LIN {X 0,Y 118.169,Z 614.006,A -85,B 0,C 180,E1 -30059.995,E2 -30059.995} C_VEL
LIN {X 0,Y 117.877,Z 614.865,A -85,B 0,C 180,E1 -30059.712,E2 -30059.712} C_VEL
LIN {X 0,Y 113.586,Z 625.245,A -85,B 0,C 180,E1 -30059.502,E2 -30059.502} C_VEL
LIN {X 0,Y 107.189,Z 637.349,A -85,B 0,C 180,E1 -30059.098,E2 -30059.098} C_VEL
LIN {X 0,Y 99.298,Z 648.743,A -85,B 0,C 180,E1 -30058.635,E2 -30058.635} C_VEL
LIN {X 0,Y 93.168,Z 656.159,A -85,B 0,C 180,E1 -30058.165,E2 -30058.165} C_VEL
LIN {X 0,Y 84.422,Z 664.947,A -85,B 0,C 180,E1 -30057.397,E2 -30057.397} C_VEL
LIN {X 0,Y 77.444,Z 670.933,A -85,B 0,C 180,E1 -30056.595,E2 -30056.595} C_VEL
LIN {X 0,Y 68.747,Z 677.24,A -85,B 0,C 180,E1 -30055.367,E2 -30055.367} C_VEL
LIN {X 0,Y 59.764,Z 682.696,A -85,B 0,C 180,E1 -30053.548,E2 -30053.548} C_VEL
LIN {X 0,Y 49.831,Z 687.613,A -85,B 0,C 180,E1 -30050.836,E2 -30050.836} C_VEL
LIN {X 0,Y 39.702,Z 691.58,A -85,B 0,C 180,E1 -30046.802,E2 -30046.802} C_VEL
LIN {X 0,Y 29.884,Z 694.52,A -85,B 0,C 180,E1 -30040.167,E2 -30040.167} C_VEL
LIN {X 0,Y 23.763,Z 696.03,A -85,B 0,C 180,E1 -30032.531,E2 -30032.531} C_VEL
LIN {X 0,Y 14.258,Z 697.578,A -85,B 0,C 180,E1 -29999.533,E2 -29999.533} C_VEL
LIN {X 0,Y 12.869,Z 697.867,A -85,B 0,C 180,E1 -29970,E2 -29970} C_VEL
LIN {X 0,Y 18.308,Z 696.97,A -85,B 0,C 180,E1 -29919.849,E2 -29919.849} C_VEL
LIN {X 0,Y 23.763,Z 696.03,A -85,B 0,C 180,E1 -29907.469,E2 -29907.469} C_VEL
LIN {X 0,Y 36.383,Z 692.67,A -85,B 0,C 180,E1 -29895.024,E2 -29895.024} C_VEL
LIN {X 0,Y 46.427,Z 689.041,A -85,B 0,C 180,E1 -29890.284,E2 -29890.284} C_VEL
LIN {X 0,Y 54.933,Z 685.21,A -85,B 0,C 180,E1 -29887.605,E2 -29887.605} C_VEL
LIN {X 0,Y 63.552,Z 680.518,A -85,B 0,C 180,E1 -29885.579,E2 -29885.579} C_VEL
LIN {X 0,Y 72.219,Z 674.865,A -85,B 0,C 180,E1 -29884.083,E2 -29884.083} C_VEL
LIN {X 0,Y 80.93,Z 668.066,A -85,B 0,C 180,E1 -29882.979,E2 -29882.979} C_VEL
LIN {X 0,Y 89.665,Z 659.854,A -85,B 0,C 180,E1 -29882.079,E2 -29882.079} C_VEL
LIN {X 0,Y 96.669,Z 652.036,A -85,B 0,C 180,E1 -29881.551,E2 -29881.551} C_VEL
LIN {X 0,Y 102.804,Z 643.959,A -85,B 0,C 180,E1 -29881.136,E2 -29881.136} C_VEL
LIN {X 0,Y 108.944,Z 634.208,A -85,B 0,C 180,E1 -29880.826,E2 -29880.826} C_VEL
LIN {X 0,Y 114.037,Z 624.239,A -85,B 0,C 180,E1 -29880.518,E2 -29880.518} C_VEL
LIN {X 0,Y 117.877,Z 614.869,A -85,B 0,C 180,E1 -29880.322,E2 -29880.322} C_VEL
LIN {X 0,Y 118.172,Z 613.998,A -85,B 0,C 180,E1 -29880.005,E2 -29880.005} C_VEL
LIN {X 0,Y 117.763,Z 615.989,A -85,B 0,C 180,E1 -29875.422,E2 -29875.422} C_VEL
LIN {X 0,Y 117.614,Z 617.596,A -85,B 0,C 180,E1 -29873.142,E2 -29873.142} C_VEL
LIN {X 0,Y 117.105,Z 620.39,A -85,B 0,C 180,E1 -29870.506,E2 -29870.506} C_VEL
LIN {X 0,Y 116.14,Z 624.865,A -85,B 0,C 180,E1 -29867.601,E2 -29867.601} C_VEL
LIN {X 0,Y 115.107,Z 628.526,A -85,B 0,C 180,E1 -29865.87,E2 -29865.87} C_VEL
LIN {X 0,Y 111.487,Z 638.971,A -85,B 0,C 180,E1 -29861.01,E2 -29861.01} C_VEL
LIN {X 0,Y 108.455,Z 647.592,A -85,B 0,C 180,E1 -29856.115,E2 -29856.115} C_VEL
LIN {X 0,Y 106.01,Z 655.467,A -85,B 0,C 180,E1 -29850.569,E2 -29850.569} C_VEL
LIN {X 0,Y 104.558,Z 661.545,A -85,B 0,C 180,E1 -29845.542,E2 -29845.542} C_VEL
LIN {X 0,Y 103.809,Z 669.53,A -85,B 0,C 180,E1 -29837.398,E2 -29837.398} C_VEL
LIN {X 0,Y 104.443,Z 673.875,A -85,B 0,C 180,E1 -29832.262,E2 -29832.262} C_VEL
LIN {X 0,Y 106.959,Z 679.238,A -85,B 0,C 180,E1 -29824.795,E2 -29824.795} C_VEL
LIN {X 0,Y 112.881,Z 684.586,A -85,B 0,C 180,E1 -29815.837,E2 -29815.837} C_VEL
LIN {X 0,Y 119.382,Z 687.768,A -85,B 0,C 180,E1 -29809.642,E2 -29809.642} C_VEL
LIN {X 0,Y 130.255,Z 690.725,A -85,B 0,C 180,E1 -29802.464,E2 -29802.464} C_VEL
LIN {X 0,Y 141.656,Z 692.301,A -85,B 0,C 180,E1 -29797.174,E2 -29797.174} C_VEL
LIN {X 0,Y 154.94,Z 692.973,A -85,B 0,C 180,E1 -29792.6,E2 -29792.6} C_VEL
LIN {X 0,Y 164.279,Z 692.971,A -85,B 0,C 180,E1 -29790,E2 -29790} C_VEL
LIN {X 0,Y 146.004,Z 692.638,A -85,B 0,C 180,E1 -29784.476,E2 -29784.476} C_VEL
LIN {X 0,Y 135.499,Z 691.643,A -85,B 0,C 180,E1 -29780.195,E2 -29780.195} C_VEL
LIN {X 0,Y 129.979,Z 690.679,A -85,B 0,C 180,E1 -29777.394,E2 -29777.394} C_VEL
LIN {X 0,Y 125.959,Z 690.113,A -85,B 0,C 180,E1 -29775.472,E2 -29775.472} C_VEL
LIN {X 0,Y 112.356,Z 688.655,A -85,B 0,C 180,E1 -29769.954,E2 -29769.954} C_VEL
LIN {X 0,Y 108.7,Z 687.726,A -85,B 0,C 180,E1 -29767.606,E2 -29767.606} C_VEL
LIN {X 0,Y 107.751,Z 687.318,A -85,B 0,C 180,E1 -29766.722,E2 -29766.722} C_VEL
LIN {X 0,Y 102.213,Z 683.666,A -85,B 0,C 180,E1 -29759.228,E2 -29759.228} C_VEL
LIN {X 0,Y 98.445,Z 678.262,A -85,B 0,C 180,E1 -29750.021,E2 -29750.021} C_VEL
LIN {X 0,Y 97.481,Z 673.186,A -85,B 0,C 180,E1 -29742.695,E2 -29742.695} C_VEL
LIN {X 0,Y 98.282,Z 666.575,A -85,B 0,C 180,E1 -29734.887,E2 -29734.887} C_VEL
LIN {X 0,Y 100.458,Z 659.553,A -85,B 0,C 180,E1 -29728.17,E2 -29728.17} C_VEL
LIN {X 0,Y 103.759,Z 651.316,A -85,B 0,C 180,E1 -29721.863,E2 -29721.863} C_VEL
LIN {X 0,Y 107.51,Z 642.683,A -85,B 0,C 180,E1 -29716.593,E2 -29716.593} C_VEL
LIN {X 0,Y 111.381,Z 633.584,A -85,B 0,C 180,E1 -29712.125,E2 -29712.125} C_VEL
LIN {X 0,Y 112.591,Z 630.569,A -85,B 0,C 180,E1 -29710.787,E2 -29710.787} C_VEL
LIN {X 0,Y 113.778,Z 627.253,A -85,B 0,C 180,E1 -29708.772,E2 -29708.772} C_VEL
LIN {X 0,Y 114.375,Z 624.991,A -85,B 0,C 180,E1 -29707.054,E2 -29707.054} C_VEL
LIN {X 0,Y 114.764,Z 623.365,A -85,B 0,C 180,E1 -29705.265,E2 -29705.265} C_VEL
LIN {X 0,Y 115.055,Z 622.207,A -85,B 0,C 180,E1 -29703.497,E2 -29703.497} C_VEL
LIN {X 0,Y 114.198,Z 624.038,A -85,B 0,C 180,E1 -29703.082,E2 -29703.082} C_VEL
LIN {X 0,Y 109.96,Z 632.42,A -85,B 0,C 180,E1 -29702.978,E2 -29702.978} C_VEL
LIN {X 0,Y 104.67,Z 641.139,A -85,B 0,C 180,E1 -29702.856,E2 -29702.856} C_VEL
LIN {X 0,Y 98.501,Z 649.644,A -85,B 0,C 180,E1 -29702.715,E2 -29702.715} C_VEL
LIN {X 0,Y 91.451,Z 657.81,A -85,B 0,C 180,E1 -29702.514,E2 -29702.514} C_VEL
LIN {X 0,Y 84.399,Z 664.75,A -85,B 0,C 180,E1 -29702.236,E2 -29702.236} C_VEL
LIN {X 0,Y 77.349,Z 670.736,A -85,B 0,C 180,E1 -29701.877,E2 -29701.877} C_VEL
LIN {X 0,Y 68.54,Z 677.044,A -85,B 0,C 180,E1 -29701.309,E2 -29701.309} C_VEL
LIN {X 0,Y 59.739,Z 682.319,A -85,B 0,C 180,E1 -29700.453,E2 -29700.453} C_VEL
LIN {X 0,Y 49.202,Z 687.416,A -85,B 0,C 180,E1 -29699.067,E2 -29699.067} C_VEL
LIN {X 0,Y 38.701,Z 691.383,A -85,B 0,C 180,E1 -29697.149,E2 -29697.149} C_VEL
LIN {X 0,Y 28.273,Z 694.323,A -85,B 0,C 180,E1 -29693.877,E2 -29693.877} C_VEL
LIN {X 0,Y 21.426,Z 695.833,A -85,B 0,C 180,E1 -29689.747,E2 -29689.747} C_VEL
LIN {X 0,Y 8.799,Z 697.381,A -85,B 0,C 180,E1 -29663.004,E2 -29663.004} C_VEL
LIN {X 0,Y 5.756,Z 697.671,A -85,B 0,C 180,E1 -29610,E2 -29610} C_VEL
LIN {X 0,Y 14.791,Z 696.773,A -85,B 0,C 180,E1 -29538.136,E2 -29538.136} C_VEL
LIN {X 0,Y 21.426,Z 695.833,A -85,B 0,C 180,E1 -29530.252,E2 -29530.252} C_VEL
LIN {X 0,Y 35.216,Z 692.474,A -85,B 0,C 180,E1 -29523.768,E2 -29523.768} C_VEL
LIN {X 0,Y 45.697,Z 688.844,A -85,B 0,C 180,E1 -29521.471,E2 -29521.471} C_VEL
LIN {X 0,Y 56.223,Z 684.109,A -85,B 0,C 180,E1 -29519.932,E2 -29519.932} C_VEL
LIN {X 0,Y 66.779,Z 678.135,A -85,B 0,C 180,E1 -29518.818,E2 -29518.818} C_VEL
LIN {X 0,Y 75.587,Z 672.046,A -85,B 0,C 180,E1 -29518.198,E2 -29518.198} C_VEL
LIN {X 0,Y 82.636,Z 666.31,A -85,B 0,C 180,E1 -29517.859,E2 -29517.859} C_VEL
LIN {X 0,Y 89.689,Z 659.658,A -85,B 0,C 180,E1 -29517.539,E2 -29517.539} C_VEL
LIN {X 0,Y 96.738,Z 651.84,A -85,B 0,C 180,E1 -29517.345,E2 -29517.345} C_VEL
LIN {X 0,Y 102.908,Z 643.763,A -85,B 0,C 180,E1 -29517.185,E2 -29517.185} C_VEL
LIN {X 0,Y 109.074,Z 634.012,A -85,B 0,C 180,E1 -29517.087,E2 -29517.087} C_VEL
LIN {X 0,Y 114.221,Z 623.981,A -85,B 0,C 180,E1 -29516.957,E2 -29516.957} C_VEL
LIN {X 0,Y 114.699,Z 622.913,A -85,B 0,C 180,E1 -29516.954,E2 -29516.954} C_VEL
LIN {X 0,Y 115.069,Z 622.175,A -85,B 0,C 180,E1 -29516.504,E2 -29516.504} C_VEL
LIN {X 0,Y 114.776,Z 623.339,A -85,B 0,C 180,E1 -29514.735,E2 -29514.735} C_VEL
LIN {X 0,Y 114.111,Z 626.031,A -85,B 0,C 180,E1 -29512.084,E2 -29512.084} C_VEL
LIN {X 0,Y 113.261,Z 628.786,A -85,B 0,C 180,E1 -29510.225,E2 -29510.225} C_VEL
LIN {X 0,Y 111.785,Z 632.565,A -85,B 0,C 180,E1 -29508.324,E2 -29508.324} C_VEL
LIN {X 0,Y 108.15,Z 641.164,A -85,B 0,C 180,E1 -29504.221,E2 -29504.221} C_VEL
LIN {X 0,Y 104.826,Z 648.774,A -85,B 0,C 180,E1 -29499.82,E2 -29499.82} C_VEL
LIN {X 0,Y 102.329,Z 654.783,A -85,B 0,C 180,E1 -29495.671,E2 -29495.671} C_VEL
LIN {X 0,Y 99.693,Z 661.815,A -85,B 0,C 180,E1 -29489.833,E2 -29489.833} C_VEL
LIN {X 0,Y 97.787,Z 669.151,A -85,B 0,C 180,E1 -29482.238,E2 -29482.238} C_VEL
LIN {X 0,Y 97.688,Z 675.553,A -85,B 0,C 180,E1 -29474.002,E2 -29474.002} C_VEL
LIN {X 0,Y 99.545,Z 680.564,A -85,B 0,C 180,E1 -29466.239,E2 -29466.239} C_VEL
LIN {X 0,Y 103.704,Z 684.913,A -85,B 0,C 180,E1 -29458.25,E2 -29458.25} C_VEL
LIN {X 0,Y 108.04,Z 687.465,A -85,B 0,C 180,E1 -29452.973,E2 -29452.973} C_VEL
LIN {X 0,Y 116.689,Z 690.455,A -85,B 0,C 180,E1 -29445.517,E2 -29445.517} C_VEL
LIN {X 0,Y 128.026,Z 692.417,A -85,B 0,C 180,E1 -29438.879,E2 -29438.879} C_VEL
LIN {X 0,Y 143.096,Z 693.294,A -85,B 0,C 180,E1 -29432.815,E2 -29432.815} C_VEL
LIN {X 0,Y 152.364,Z 693.301,A -85,B 0,C 180,E1 -29430,E2 -29430} C_VEL
LIN {X 0,Y 140.823,Z 693.282,A -85,B 0,C 180,E1 -29426.413,E2 -29426.413} C_VEL
LIN {X 0,Y 126.564,Z 692.278,A -85,B 0,C 180,E1 -29420.411,E2 -29420.411} C_VEL
LIN {X 0,Y 116.678,Z 690.465,A -85,B 0,C 180,E1 -29414.503,E2 -29414.503} C_VEL
LIN {X 0,Y 107.751,Z 687.318,A -85,B 0,C 180,E1 -29406.722,E2 -29406.722} C_VEL
LIN {X 0,Y 104.734,Z 686.184,A -85,B 0,C 180,E1 -29404.045,E2 -29404.045} C_VEL
LIN {X 0,Y 94.611,Z 683.451,A -85,B 0,C 180,E1 -29395.741,E2 -29395.741} C_VEL
LIN {X 0,Y 92.503,Z 682.035,A -85,B 0,C 180,E1 -29392.488,E2 -29392.488} C_VEL
LIN {X 0,Y 92.124,Z 681.457,A -85,B 0,C 180,E1 -29391.348,E2 -29391.348} C_VEL
LIN {X 0,Y 91.057,Z 677.2,A -85,B 0,C 180,E1 -29383.988,E2 -29383.988} C_VEL
LIN {X 0,Y 91.647,Z 671.97,A -85,B 0,C 180,E1 -29376.453,E2 -29376.453} C_VEL
LIN {X 0,Y 93.783,Z 665.721,A -85,B 0,C 180,E1 -29369.14,E2 -29369.14} C_VEL
LIN {X 0,Y 96.531,Z 659.898,A -85,B 0,C 180,E1 -29363.595,E2 -29363.595} C_VEL
LIN {X 0,Y 100.499,Z 652.251,A -85,B 0,C 180,E1 -29357.733,E2 -29357.733} C_VEL
LIN {X 0,Y 104.974,Z 643.783,A -85,B 0,C 180,E1 -29352.617,E2 -29352.617} C_VEL
LIN {X 0,Y 109.775,Z 634.122,A -85,B 0,C 180,E1 -29347.933,E2 -29347.933} C_VEL
LIN {X 0,Y 110.243,Z 633.033,A -85,B 0,C 180,E1 -29347.319,E2 -29347.319} C_VEL
LIN {X 0,Y 109.183,Z 634.691,A -85,B 0,C 180,E1 -29346.655,E2 -29346.655} C_VEL
LIN {X 0,Y 101.738,Z 646.132,A -85,B 0,C 180,E1 -29346.782,E2 -29346.782} C_VEL
LIN {X 0,Y 93.799,Z 655.765,A -85,B 0,C 180,E1 -29346.899,E2 -29346.899} C_VEL
LIN {X 0,Y 84.976,Z 664.553,A -85,B 0,C 180,E1 -29347.041,E2 -29347.041} C_VEL
LIN {X 0,Y 77.909,Z 670.539,A -85,B 0,C 180,E1 -29347.126,E2 -29347.126} C_VEL
LIN {X 0,Y 69.072,Z 676.846,A -85,B 0,C 180,E1 -29347.236,E2 -29347.236} C_VEL
LIN {X 0,Y 60.223,Z 682.121,A -85,B 0,C 180,E1 -29347.28,E2 -29347.28} C_VEL
LIN {X 0,Y 49.602,Z 687.219,A -85,B 0,C 180,E1 -29347.337,E2 -29347.337} C_VEL
LIN {X 0,Y 39.005,Z 691.185,A -85,B 0,C 180,E1 -29347.697,E2 -29347.697} C_VEL
LIN {X 0,Y 28.409,Z 694.126,A -85,B 0,C 180,E1 -29348.301,E2 -29348.301} C_VEL
LIN {X 0,Y 21.345,Z 695.635,A -85,B 0,C 180,E1 -29348.978,E2 -29348.978} C_VEL
LIN {X 0,Y 7.264,Z 697.184,A -85,B 0,C 180,E1 -29354.645,E2 -29354.645} C_VEL
LIN {X 0,Y 1.343,Z 697.475,A -85,B 0,C 180,E1 -29430,E2 -29430} C_VEL
LIN {X 0,Y 14.283,Z 696.575,A -85,B 0,C 180,E1 -29509.759,E2 -29509.759} C_VEL
LIN {X 0,Y 21.345,Z 695.635,A -85,B 0,C 180,E1 -29511.022,E2 -29511.022} C_VEL
LIN {X 0,Y 35.466,Z 692.277,A -85,B 0,C 180,E1 -29512.216,E2 -29512.216} C_VEL
LIN {X 0,Y 46.066,Z 688.647,A -85,B 0,C 180,E1 -29512.589,E2 -29512.589} C_VEL
LIN {X 0,Y 55.231,Z 684.646,A -85,B 0,C 180,E1 -29512.701,E2 -29512.701} C_VEL
LIN {X 0,Y 65.538,Z 679.03,A -85,B 0,C 180,E1 -29512.713,E2 -29512.713} C_VEL
LIN {X 0,Y 74.378,Z 673.16,A -85,B 0,C 180,E1 -29512.813,E2 -29512.813} C_VEL
LIN {X 0,Y 81.441,Z 667.673,A -85,B 0,C 180,E1 -29512.927,E2 -29512.927} C_VEL
LIN {X 0,Y 90.272,Z 659.462,A -85,B 0,C 180,E1 -29513.035,E2 -29513.035} C_VEL
LIN {X 0,Y 97.326,Z 651.643,A -85,B 0,C 180,E1 -29513.161,E2 -29513.161} C_VEL
LIN {X 0,Y 103.498,Z 643.567,A -85,B 0,C 180,E1 -29513.262,E2 -29513.262} C_VEL
LIN {X 0,Y 109.172,Z 634.704,A -85,B 0,C 180,E1 -29513.368,E2 -29513.368} C_VEL
LIN {X 0,Y 110.22,Z 633.075,A -85,B 0,C 180,E1 -29512.679,E2 -29512.679} C_VEL
LIN {X 0,Y 107.201,Z 639.436,A -85,B 0,C 180,E1 -29509.539,E2 -29509.539} C_VEL
LIN {X 0,Y 102.878,Z 647.758,A -85,B 0,C 180,E1 -29505.104,E2 -29505.104} C_VEL
LIN {X 0,Y 99.152,Z 654.795,A -85,B 0,C 180,E1 -29500.508,E2 -29500.508} C_VEL
LIN {X 0,Y 95.086,Z 662.884,A -85,B 0,C 180,E1 -29493.682,E2 -29493.682} C_VEL
LIN {X 0,Y 92.412,Z 669.407,A -85,B 0,C 180,E1 -29486.777,E2 -29486.777} C_VEL
LIN {X 0,Y 91.145,Z 675.365,A -85,B 0,C 180,E1 -29478.846,E2 -29478.846} C_VEL
LIN {X 0,Y 91.811,Z 680.718,A -85,B 0,C 180,E1 -29470.061,E2 -29470.061} C_VEL
LIN {X 0,Y 94.843,Z 685.153,A -85,B 0,C 180,E1 -29461.245,E2 -29461.245} C_VEL
LIN {X 0,Y 99.773,Z 688.355,A -85,B 0,C 180,E1 -29453.709,E2 -29453.709} C_VEL
LIN {X 0,Y 109.071,Z 691.344,A -85,B 0,C 180,E1 -29444.891,E2 -29444.891} C_VEL
LIN {X 0,Y 115.719,Z 692.583,A -85,B 0,C 180,E1 -29440.498,E2 -29440.498} C_VEL
LIN {X 0,Y 126.949,Z 693.553,A -85,B 0,C 180,E1 -29434.865,E2 -29434.865} C_VEL
LIN {X 0,Y 140.481,Z 693.629,A -85,B 0,C 180,E1 -29430,E2 -29430} C_VEL
LIN {X 0,Y 126.947,Z 693.555,A -85,B 0,C 180,E1 -29425.143,E2 -29425.143} C_VEL
LIN {X 0,Y 114.594,Z 692.424,A -85,B 0,C 180,E1 -29418.861,E2 -29418.861} C_VEL
LIN {X 0,Y 103.287,Z 689.725,A -85,B 0,C 180,E1 -29410.11,E2 -29410.11} C_VEL
LIN {X 0,Y 98.564,Z 687.752,A -85,B 0,C 180,E1 -29404.671,E2 -29404.671} C_VEL
LIN {X 0,Y 93.554,Z 683.757,A -85,B 0,C 180,E1 -29395.713,E2 -29395.713} C_VEL
LIN {X 0,Y 92.124,Z 681.457,A -85,B 0,C 180,E1 -29391.348,E2 -29391.348} C_VEL
LIN {X 0,Y 90.843,Z 679.857,A -85,B 0,C 180,E1 -29387.872,E2 -29387.872} C_VEL
LIN {X 0,Y 86.151,Z 675.628,A -85,B 0,C 180,E1 -29377.053,E2 -29377.053} C_VEL
LIN {X 0,Y 86,Z 673.585,A -85,B 0,C 180,E1 -29373.388,E2 -29373.388} C_VEL
LIN {X 0,Y 86.266,Z 672.75,A -85,B 0,C 180,E1 -29372.221,E2 -29372.221} C_VEL
LIN {X 0,Y 89.365,Z 666.65,A -85,B 0,C 180,E1 -29364.808,E2 -29364.808} C_VEL
LIN {X 0,Y 93.127,Z 660.513,A -85,B 0,C 180,E1 -29358.914,E2 -29358.914} C_VEL
LIN {X 0,Y 98.879,Z 651.385,A -85,B 0,C 180,E1 -29352.234,E2 -29352.234} C_VEL
LIN {X 0,Y 100.187,Z 649.251,A -85,B 0,C 180,E1 -29350.867,E2 -29350.867} C_VEL
LIN {X 0,Y 93.162,Z 657.417,A -85,B 0,C 180,E1 -29351.278,E2 -29351.278} C_VEL
LIN {X 0,Y 86.139,Z 664.356,A -85,B 0,C 180,E1 -29351.747,E2 -29351.747} C_VEL
LIN {X 0,Y 79.108,Z 670.342,A -85,B 0,C 180,E1 -29352.248,E2 -29352.248} C_VEL
LIN {X 0,Y 70.325,Z 676.65,A -85,B 0,C 180,E1 -29353.002,E2 -29353.002} C_VEL
LIN {X 0,Y 61.537,Z 681.924,A -85,B 0,C 180,E1 -29353.892,E2 -29353.892} C_VEL
LIN {X 0,Y 51.01,Z 687.021,A -85,B 0,C 180,E1 -29355.327,E2 -29355.327} C_VEL
LIN {X 0,Y 40.584,Z 690.988,A -85,B 0,C 180,E1 -29357.742,E2 -29357.742} C_VEL
LIN {X 0,Y 30.266,Z 693.93,A -85,B 0,C 180,E1 -29361.747,E2 -29361.747} C_VEL
LIN {X 0,Y 23.541,Z 695.438,A -85,B 0,C 180,E1 -29366.414,E2 -29366.414} C_VEL
LIN {X 0,Y 11.387,Z 696.987,A -85,B 0,C 180,E1 -29391.89,E2 -29391.89} C_VEL
LIN {X 0,Y 8.433,Z 697.279,A -85,B 0,C 180,E1 -29430,E2 -29430} C_VEL
LIN {X 0,Y 17.064,Z 696.378,A -85,B 0,C 180,E1 -29485.457,E2 -29485.457} C_VEL
LIN {X 0,Y 23.542,Z 695.438,A -85,B 0,C 180,E1 -29493.585,E2 -29493.585} C_VEL
LIN {X 0,Y 37.113,Z 692.08,A -85,B 0,C 180,E1 -29501.231,E2 -29501.231} C_VEL
LIN {X 0,Y 47.512,Z 688.451,A -85,B 0,C 180,E1 -29504.046,E2 -29504.046} C_VEL
LIN {X 0,Y 55.54,Z 684.983,A -85,B 0,C 180,E1 -29505.352,E2 -29505.352} C_VEL
LIN {X 0,Y 66.815,Z 678.834,A -85,B 0,C 180,E1 -29506.646,E2 -29506.646} C_VEL
LIN {X 0,Y 75.601,Z 672.963,A -85,B 0,C 180,E1 -29507.444,E2 -29507.444} C_VEL
LIN {X 0,Y 82.617,Z 667.476,A -85,B 0,C 180,E1 -29508.032,E2 -29508.032} C_VEL
LIN {X 0,Y 91.409,Z 659.265,A -85,B 0,C 180,E1 -29508.6,E2 -29508.6} C_VEL
LIN {X 0,Y 98.427,Z 651.447,A -85,B 0,C 180,E1 -29509.046,E2 -29509.046} C_VEL
LIN {X 0,Y 100.215,Z 649.247,A -85,B 0,C 180,E1 -29509.05,E2 -29509.05} C_VEL
LIN {X 0,Y 95.856,Z 656.134,A -85,B 0,C 180,E1 -29504.553,E2 -29504.553} C_VEL
LIN {X 0,Y 90.993,Z 663.897,A -85,B 0,C 180,E1 -29497.947,E2 -29497.947} C_VEL
LIN {X 0,Y 87.501,Z 670.11,A -85,B 0,C 180,E1 -29491.198,E2 -29491.198} C_VEL
LIN {X 0,Y 85.508,Z 674.843,A -85,B 0,C 180,E1 -29484.886,E2 -29484.886} C_VEL
LIN {X 0,Y 84.56,Z 680.62,A -85,B 0,C 180,E1 -29475.064,E2 -29475.064} C_VEL
LIN {X 0,Y 86.454,Z 685.429,A -85,B 0,C 180,E1 -29464.683,E2 -29464.683} C_VEL
LIN {X 0,Y 89.357,Z 688.037,A -85,B 0,C 180,E1 -29458.158,E2 -29458.158} C_VEL
LIN {X 0,Y 96.479,Z 691.081,A -85,B 0,C 180,E1 -29448.762,E2 -29448.762} C_VEL
LIN {X 0,Y 107.096,Z 693.104,A -85,B 0,C 180,E1 -29440.186,E2 -29440.186} C_VEL
LIN {X 0,Y 120.064,Z 693.922,A -85,B 0,C 180,E1 -29433.356,E2 -29433.356} C_VEL
LIN {X 0,Y 128.809,Z 693.952,A -85,B 0,C 180,E1 -29430,E2 -29430} C_VEL
LIN {X 0,Y 113.19,Z 693.668,A -85,B 0,C 180,E1 -29423.383,E2 -29423.383} C_VEL
LIN {X 0,Y 104.921,Z 692.887,A -85,B 0,C 180,E1 -29418.408,E2 -29418.408} C_VEL
LIN {X 0,Y 96.479,Z 691.081,A -85,B 0,C 180,E1 -29411.237,E2 -29411.237} C_VEL
LIN {X 0,Y 88.743,Z 687.517,A -85,B 0,C 180,E1 -29400.577,E2 -29400.577} C_VEL
LIN {X 0,Y 85.418,Z 683.748,A -85,B 0,C 180,E1 -29391.394,E2 -29391.394} C_VEL
LIN {X 0,Y 84.572,Z 678.795,A -85,B 0,C 180,E1 -29381.592,E2 -29381.592} C_VEL
LIN {X 0,Y 86.266,Z 672.75,A -85,B 0,C 180,E1 -29372.221,E2 -29372.221} C_VEL
LIN {X 0,Y 86.512,Z 671.274,A -85,B 0,C 180,E1 -29369.764,E2 -29369.764} C_VEL
LIN {X 0,Y 85.588,Z 667.944,A -85,B 0,C 180,E1 -29361.065,E2 -29361.065} C_VEL
LIN {X 0,Y 86.473,Z 666.237,A -85,B 0,C 180,E1 -29358.738,E2 -29358.738} C_VEL
LIN {X 0,Y 88.039,Z 664.142,A -85,B 0,C 180,E1 -29356.68,E2 -29356.68} C_VEL
LIN {X 0,Y 87.862,Z 664.16,A -85,B 0,C 180,E1 -29356.289,E2 -29356.289} C_VEL
LIN {X 0,Y 80.916,Z 670.146,A -85,B 0,C 180,E1 -29357.176,E2 -29357.176} C_VEL
LIN {X 0,Y 72.266,Z 676.452,A -85,B 0,C 180,E1 -29358.524,E2 -29358.524} C_VEL
LIN {X 0,Y 63.633,Z 681.726,A -85,B 0,C 180,E1 -29360.153,E2 -29360.153} C_VEL
LIN {X 0,Y 53.345,Z 686.824,A -85,B 0,C 180,E1 -29362.748,E2 -29362.748} C_VEL
LIN {X 0,Y 43.294,Z 690.79,A -85,B 0,C 180,E1 -29366.77,E2 -29366.77} C_VEL
LIN {X 0,Y 33.556,Z 693.733,A -85,B 0,C 180,E1 -29373.097,E2 -29373.097} C_VEL
LIN {X 0,Y 27.471,Z 695.24,A -85,B 0,C 180,E1 -29379.872,E2 -29379.872} C_VEL
LIN {X 0,Y 17.543,Z 696.791,A -85,B 0,C 180,E1 -29406.384,E2 -29406.384} C_VEL
LIN {X 0,Y 15.542,Z 697.082,A -85,B 0,C 180,E1 -29430,E2 -29430} C_VEL
LIN {X 0,Y 21.908,Z 696.181,A -85,B 0,C 180,E1 -29469.911,E2 -29469.911} C_VEL
LIN {X 0,Y 27.471,Z 695.24,A -85,B 0,C 180,E1 -29480.128,E2 -29480.128} C_VEL
LIN {X 0,Y 39.991,Z 691.882,A -85,B 0,C 180,E1 -29491.484,E2 -29491.484} C_VEL
LIN {X 0,Y 49.95,Z 688.253,A -85,B 0,C 180,E1 -29496.142,E2 -29496.142} C_VEL
LIN {X 0,Y 60.19,Z 683.517,A -85,B 0,C 180,E1 -29499.082,E2 -29499.082} C_VEL
LIN {X 0,Y 70.537,Z 677.545,A -85,B 0,C 180,E1 -29501.178,E2 -29501.178} C_VEL
LIN {X 0,Y 79.19,Z 671.456,A -85,B 0,C 180,E1 -29502.562,E2 -29502.562} C_VEL
LIN {X 0,Y 85.712,Z 666.088,A -85,B 0,C 180,E1 -29503.452,E2 -29503.452} C_VEL
LIN {X 0,Y 87.861,Z 664.16,A -85,B 0,C 180,E1 -29503.712,E2 -29503.712} C_VEL
LIN {X 0,Y 88.039,Z 664.143,A -85,B 0,C 180,E1 -29503.322,E2 -29503.322} C_VEL
LIN {X 0,Y 83.847,Z 669.909,A -85,B 0,C 180,E1 -29497.22,E2 -29497.22} C_VEL
LIN {X 0,Y 79.779,Z 676.411,A -85,B 0,C 180,E1 -29488.102,E2 -29488.102} C_VEL
LIN {X 0,Y 78.039,Z 681.486,A -85,B 0,C 180,E1 -29478.662,E2 -29478.662} C_VEL
LIN {X 0,Y 78.573,Z 685.701,A -85,B 0,C 180,E1 -29468.764,E2 -29468.764} C_VEL
LIN {X 0,Y 81.215,Z 688.752,A -85,B 0,C 180,E1 -29460.093,E2 -29460.093} C_VEL
LIN {X 0,Y 84.533,Z 690.555,A -85,B 0,C 180,E1 -29453.881,E2 -29453.881} C_VEL
LIN {X 0,Y 94.469,Z 693.182,A -85,B 0,C 180,E1 -29442.896,E2 -29442.896} C_VEL
LIN {X 0,Y 108.891,Z 694.232,A -85,B 0,C 180,E1 -29433.7,E2 -29433.7} C_VEL
LIN {X 0,Y 117.313,Z 694.269,A -85,B 0,C 180,E1 -29430,E2 -29430} C_VEL
LIN {X 0,Y 105.853,Z 694.207,A -85,B 0,C 180,E1 -29424.741,E2 -29424.741} C_VEL
LIN {X 0,Y 93.894,Z 693.094,A -85,B 0,C 180,E1 -29416.638,E2 -29416.638} C_VEL
LIN {X 0,Y 84.059,Z 690.299,A -85,B 0,C 180,E1 -29405.289,E2 -29405.289} C_VEL
LIN {X 0,Y 80.697,Z 688.313,A -85,B 0,C 180,E1 -29398.497,E2 -29398.497} C_VEL
LIN {X 0,Y 77.969,Z 683.667,A -85,B 0,C 180,E1 -29386.133,E2 -29386.133} C_VEL
LIN {X 0,Y 78.844,Z 678.402,A -85,B 0,C 180,E1 -29375.283,E2 -29375.283} C_VEL
LIN {X 0,Y 81.805,Z 672.898,A -85,B 0,C 180,E1 -29366.628,E2 -29366.628} C_VEL
LIN {X 0,Y 86.473,Z 666.237,A -85,B 0,C 180,E1 -29358.738,E2 -29358.738} C_VEL
LIN {X 0,Y 85.989,Z 666.47,A -85,B 0,C 180,E1 -29358.239,E2 -29358.239} C_VEL
LIN {X 0,Y 84.009,Z 668.065,A -85,B 0,C 180,E1 -29358.045,E2 -29358.045} C_VEL
LIN {X 0,Y 80.183,Z 671.177,A -85,B 0,C 180,E1 -29358.876,E2 -29358.876} C_VEL
LIN {X 0,Y 74.975,Z 675.481,A -85,B 0,C 180,E1 -29361.196,E2 -29361.196} C_VEL
LIN {X 0,Y 70.97,Z 678.378,A -85,B 0,C 180,E1 -29363.306,E2 -29363.306} C_VEL
LIN {X 0,Y 65.72,Z 681.88,A -85,B 0,C 180,E1 -29365.904,E2 -29365.904} C_VEL
LIN {X 0,Y 62.303,Z 683.739,A -85,B 0,C 180,E1 -29367.227,E2 -29367.227} C_VEL
LIN {X 0,Y 53.234,Z 688.056,A -85,B 0,C 180,E1 -29370.894,E2 -29370.894} C_VEL
LIN {X 0,Y 43.855,Z 691.685,A -85,B 0,C 180,E1 -29376.749,E2 -29376.749} C_VEL
LIN {X 0,Y 32.51,Z 695.043,A -85,B 0,C 180,E1 -29389.569,E2 -29389.569} C_VEL
LIN {X 0,Y 24.25,Z 696.593,A -85,B 0,C 180,E1 -29413.154,E2 -29413.154} C_VEL
LIN {X 0,Y 22.64,Z 696.886,A -85,B 0,C 180,E1 -29430,E2 -29430} C_VEL
LIN {X 0,Y 27.749,Z 695.984,A -85,B 0,C 180,E1 -29460.433,E2 -29460.433} C_VEL
LIN {X 0,Y 32.51,Z 695.043,A -85,B 0,C 180,E1 -29470.431,E2 -29470.431} C_VEL
LIN {X 0,Y 43.855,Z 691.685,A -85,B 0,C 180,E1 -29483.252,E2 -29483.252} C_VEL
LIN {X 0,Y 53.241,Z 688.056,A -85,B 0,C 180,E1 -29489.095,E2 -29489.095} C_VEL
LIN {X 0,Y 61.039,Z 684.426,A -85,B 0,C 180,E1 -29492.32,E2 -29492.32} C_VEL
LIN {X 0,Y 71.598,Z 678.351,A -85,B 0,C 180,E1 -29495.5,E2 -29495.5} C_VEL
LIN {X 0,Y 76.518,Z 675.149,A -85,B 0,C 180,E1 -29496.703,E2 -29496.703} C_VEL
LIN {X 0,Y 72.132,Z 681.778,A -85,B 0,C 180,E1 -29484.236,E2 -29484.236} C_VEL
LIN {X 0,Y 71.225,Z 685.97,A -85,B 0,C 180,E1 -29473.686,E2 -29473.686} C_VEL
LIN {X 0,Y 72.377,Z 688.588,A -85,B 0,C 180,E1 -29465.634,E2 -29465.634} C_VEL
LIN {X 0,Y 76.926,Z 691.599,A -85,B 0,C 180,E1 -29454.013,E2 -29454.013} C_VEL
LIN {X 0,Y 86.343,Z 693.736,A -85,B 0,C 180,E1 -29442.415,E2 -29442.415} C_VEL
LIN {X 0,Y 98.59,Z 694.541,A -85,B 0,C 180,E1 -29433.742,E2 -29433.742} C_VEL
LIN {X 0,Y 106.034,Z 694.581,A -85,B 0,C 180,E1 -29430,E2 -29430} C_VEL
LIN {X 0,Y 90.5,Z 694.175,A -85,B 0,C 180,E1 -29421.065,E2 -29421.065} C_VEL
LIN {X 0,Y 81.208,Z 692.798,A -85,B 0,C 180,E1 -29412.144,E2 -29412.144} C_VEL
LIN {X 0,Y 74.962,Z 690.58,A -85,B 0,C 180,E1 -29402.046,E2 -29402.046} C_VEL
LIN {X 0,Y 71.771,Z 687.685,A -85,B 0,C 180,E1 -29391.556,E2 -29391.556} C_VEL
LIN {X 0,Y 71.375,Z 683.795,A -85,B 0,C 180,E1 -29380.444,E2 -29380.444} C_VEL
LIN {X 0,Y 73.457,Z 679.315,A -85,B 0,C 180,E1 -29370.564,E2 -29370.564} C_VEL
LIN {X 0,Y 76.515,Z 675.149,A -85,B 0,C 180,E1 -29363.292,E2 -29363.292} C_VEL
LIN {X 0,Y 66.422,Z 681.529,A -85,B 0,C 180,E1 -29365.927,E2 -29365.927} C_VEL
LIN {X 0,Y 62.303,Z 683.739,A -85,B 0,C 180,E1 -29367.227,E2 -29367.227} C_VEL
LIN {X 0,Y 57.598,Z 686.295,A -85,B 0,C 180,E1 -29369.647,E2 -29369.647} C_VEL
LIN {X 0,Y 50.981,Z 689.781,A -85,B 0,C 180,E1 -29376.538,E2 -29376.538} C_VEL
LIN {X 0,Y 46.334,Z 692.03,A -85,B 0,C 180,E1 -29383.704,E2 -29383.704} C_VEL
LIN {X 0,Y 42.722,Z 693.424,A -85,B 0,C 180,E1 -29389.482,E2 -29389.482} C_VEL
LIN {X 0,Y 41.408,Z 693.828,A -85,B 0,C 180,E1 -29391.407,E2 -29391.407} C_VEL
LIN {X 0,Y 38.223,Z 694.846,A -85,B 0,C 180,E1 -29396.523,E2 -29396.523} C_VEL
LIN {X 0,Y 31.137,Z 696.396,A -85,B 0,C 180,E1 -29416.956,E2 -29416.956} C_VEL
LIN {X 0,Y 29.755,Z 696.689,A -85,B 0,C 180,E1 -29430,E2 -29430} C_VEL
LIN {X 0,Y 34.093,Z 695.787,A -85,B 0,C 180,E1 -29454.348,E2 -29454.348} C_VEL
LIN {X 0,Y 38.223,Z 694.846,A -85,B 0,C 180,E1 -29463.477,E2 -29463.477} C_VEL
LIN {X 0,Y 48.467,Z 691.487,A -85,B 0,C 180,E1 -29476.471,E2 -29476.471} C_VEL
LIN {X 0,Y 57.235,Z 687.858,A -85,B 0,C 180,E1 -29482.953,E2 -29482.953} C_VEL
LIN {X 0,Y 61.815,Z 685.75,A -85,B 0,C 180,E1 -29485.369,E2 -29485.369} C_VEL
LIN {X 0,Y 65.716,Z 684.005,A -85,B 0,C 180,E1 -29485.907,E2 -29485.907} C_VEL
LIN {X 0,Y 64.669,Z 688.92,A -85,B 0,C 180,E1 -29470.487,E2 -29470.487} C_VEL
LIN {X 0,Y 66.251,Z 690.88,A -85,B 0,C 180,E1 -29461.953,E2 -29461.953} C_VEL
LIN {X 0,Y 74.133,Z 693.763,A -85,B 0,C 180,E1 -29446.523,E2 -29446.523} C_VEL
LIN {X 0,Y 87.084,Z 694.836,A -85,B 0,C 180,E1 -29434.629,E2 -29434.629} C_VEL
LIN {X 0,Y 94.956,Z 694.887,A -85,B 0,C 180,E1 -29430,E2 -29430} C_VEL
LIN {X 0,Y 84.815,Z 694.815,A -85,B 0,C 180,E1 -29423.832,E2 -29423.832} C_VEL
LIN {X 0,Y 73.585,Z 693.649,A -85,B 0,C 180,E1 -29412.731,E2 -29412.731} C_VEL
LIN {X 0,Y 66.292,Z 690.856,A -85,B 0,C 180,E1 -29397.99,E2 -29397.99} C_VEL
LIN {X 0,Y 64.647,Z 688.86,A -85,B 0,C 180,E1 -29389.287,E2 -29389.287} C_VEL
LIN {X 0,Y 65.625,Z 684.057,A -85,B 0,C 180,E1 -29374.134,E2 -29374.134} C_VEL
LIN {X 0,Y 62.387,Z 685.459,A -85,B 0,C 180,E1 -29374.269,E2 -29374.269} C_VEL
LIN {X 0,Y 54.21,Z 689.273,A -85,B 0,C 180,E1 -29378.936,E2 -29378.936} C_VEL
LIN {X 0,Y 43.044,Z 693.339,A -85,B 0,C 180,E1 -29389.225,E2 -29389.225} C_VEL
LIN {X 0,Y 41.408,Z 693.828,A -85,B 0,C 180,E1 -29391.407,E2 -29391.407} C_VEL
LIN {X 0,Y 38.056,Z 694.985,A -85,B 0,C 180,E1 -29398.263,E2 -29398.263} C_VEL
LIN {X 0,Y 35.645,Z 696.14,A -85,B 0,C 180,E1 -29413.136,E2 -29413.136} C_VEL
LIN {X 0,Y 36.824,Z 696.459,A -85,B 0,C 180,E1 -29432.124,E2 -29432.124} C_VEL
LIN {X 0,Y 37.694,Z 696.27,A -85,B 0,C 180,E1 -29438.125,E2 -29438.125} C_VEL
LIN {X 0,Y 40.693,Z 695.59,A -85,B 0,C 180,E1 -29450.207,E2 -29450.207} C_VEL
LIN {X 0,Y 44.347,Z 694.649,A -85,B 0,C 180,E1 -29458.387,E2 -29458.387} C_VEL
LIN {X 0,Y 53.631,Z 691.29,A -85,B 0,C 180,E1 -29470.935,E2 -29470.935} C_VEL
LIN {X 0,Y 57.598,Z 689.982,A -85,B 0,C 180,E1 -29472.953,E2 -29472.953} C_VEL
LIN {X 0,Y 58.832,Z 691.924,A -85,B 0,C 180,E1 -29463.278,E2 -29463.278} C_VEL
LIN {X 0,Y 65.971,Z 694.29,A -85,B 0,C 180,E1 -29446.544,E2 -29446.544} C_VEL
LIN {X 0,Y 76.413,Z 695.132,A -85,B 0,C 180,E1 -29435.277,E2 -29435.277} C_VEL
LIN {X 0,Y 84.029,Z 695.189,A -85,B 0,C 180,E1 -29430,E2 -29430} C_VEL
LIN {X 0,Y 69.789,Z 694.756,A -85,B 0,C 180,E1 -29418.381,E2 -29418.381} C_VEL
LIN {X 0,Y 64.399,Z 694.045,A -85,B 0,C 180,E1 -29410.889,E2 -29410.889} C_VEL
LIN {X 0,Y 58.842,Z 691.919,A -85,B 0,C 180,E1 -29396.707,E2 -29396.707} C_VEL
LIN {X 0,Y 57.616,Z 689.974,A -85,B 0,C 180,E1 -29387.028,E2 -29387.028} C_VEL
LIN {X 0,Y 53.632,Z 691.29,A -85,B 0,C 180,E1 -29389.065,E2 -29389.065} C_VEL
LIN {X 0,Y 44.347,Z 694.649,A -85,B 0,C 180,E1 -29401.613,E2 -29401.613} C_VEL
LIN {X 0,Y 38.104,Z 696.2,A -85,B 0,C 180,E1 -29419.371,E2 -29419.371} C_VEL
LIN {X 0,Y 36.859,Z 696.493,A -85,B 0,C 180,E1 -29430,E2 -29430} C_VEL
LIN {X 0,Y 37.694,Z 696.27,A -85,B 0,C 180,E1 -29438.125,E2 -29438.125} C_VEL
LIN {X 0,Y 39.316,Z 696.098,A -85,B 0,C 180,E1 -29443.458,E2 -29443.458} C_VEL
LIN {X 0,Y 41.973,Z 695.755,A -85,B 0,C 180,E1 -29447.61,E2 -29447.61} C_VEL
LIN {X 0,Y 50.98,Z 694.375,A -85,B 0,C 180,E1 -29454.966,E2 -29454.966} C_VEL
LIN {X 0,Y 53.218,Z 693.849,A -85,B 0,C 180,E1 -29456.603,E2 -29456.603} C_VEL
LIN {X 0,Y 59.675,Z 695.043,A -85,B 0,C 180,E1 -29443.624,E2 -29443.624} C_VEL
LIN {X 0,Y 70.323,Z 695.475,A -85,B 0,C 180,E1 -29432.251,E2 -29432.251} C_VEL
LIN {X 0,Y 73.261,Z 695.487,A -85,B 0,C 180,E1 -29430,E2 -29430} C_VEL
LIN {X 0,Y 63.901,Z 695.396,A -85,B 0,C 180,E1 -29421.754,E2 -29421.754} C_VEL
LIN {X 0,Y 54.124,Z 694.075,A -85,B 0,C 180,E1 -29405.332,E2 -29405.332} C_VEL
LIN {X 0,Y 53.379,Z 693.805,A -85,B 0,C 180,E1 -29403.24,E2 -29403.24} C_VEL
LIN {X 0,Y 50.729,Z 694.452,A -85,B 0,C 180,E1 -29405.442,E2 -29405.442} C_VEL
LIN {X 0,Y 45.109,Z 696.003,A -85,B 0,C 180,E1 -29421.037,E2 -29421.037} C_VEL
LIN {X 0,Y 43.955,Z 696.297,A -85,B 0,C 180,E1 -29430,E2 -29430} C_VEL
LIN {X 0,Y 47.465,Z 695.392,A -85,B 0,C 180,E1 -29447.225,E2 -29447.225} C_VEL
LIN {X 0,Y 50.729,Z 694.452,A -85,B 0,C 180,E1 -29454.558,E2 -29454.558} C_VEL
LIN {X 0,Y 53.218,Z 693.849,A -85,B 0,C 180,E1 -29456.603,E2 -29456.603} C_VEL
LIN {X 0,Y 54.18,Z 693.836,A -85,B 0,C 180,E1 -29456.065,E2 -29456.065} C_VEL
LIN {X 0,Y 54.814,Z 694.127,A -85,B 0,C 180,E1 -29453.925,E2 -29453.925} C_VEL
LIN {X 0,Y 54.925,Z 694.641,A -85,B 0,C 180,E1 -29449.716,E2 -29449.716} C_VEL
LIN {X 0,Y 55.13,Z 695.628,A -85,B 0,C 180,E1 -29439.964,E2 -29439.964} C_VEL
LIN {X 0,Y 56.959,Z 695.727,A -85,B 0,C 180,E1 -29435.7,E2 -29435.7} C_VEL
LIN {X 0,Y 57.536,Z 695.733,A -85,B 0,C 180,E1 -29434.995,E2 -29434.995} C_VEL
LIN {X 0,Y 62.776,Z 695.777,A -85,B 0,C 180,E1 -29430,E2 -29430} C_VEL
LIN {X 0,Y 54.153,Z 695.687,A -85,B 0,C 180,E1 -29420.78,E2 -29420.78} C_VEL
LIN {X 0,Y 52.175,Z 695.806,A -85,B 0,C 180,E1 -29422.259,E2 -29422.259} C_VEL
LIN {X 0,Y 51.078,Z 696.1,A -85,B 0,C 180,E1 -29430,E2 -29430} C_VEL
LIN {X 0,Y 52.198,Z 695.805,A -85,B 0,C 180,E1 -29437.738,E2 -29437.738} C_VEL
LIN {X 0,Y 54.143,Z 695.689,A -85,B 0,C 180,E1 -29439.179,E2 -29439.179} C_VEL
LIN {X 0,Y 57.536,Z 695.733,A -85,B 0,C 180,E1 -29434.995,E2 -29434.995} C_VEL
LIN {X 0,Y 57.536,Z 695.733,A -85,B 0,C 180,E1 -29434.995,E2 -29434.995}

QRS_NEXT_CUT()

QRS_NEXT()
QRS_HOME()

END
